(*

## Short summary

This class implements the breadth first iteration strategy for balanced binary search trees.

.. <legal notes>

legal notes
=================
| SPDX-FileCopyrightText: © 2024 ekvip automation GmbH <info@ekvip.de>
| SPDX-License-Identifier: Apache-2.0
| For details check: Apache-2.0_

.. _Apache-2.0: https://www.apache.org/licenses/LICENSE-2.0

.. </legal notes>

*)

{attribute 'enable_dynamic_creation'}
FUNCTION_BLOCK BfsBbstIterator EXTENDS AbstractBalancedBinarySearchTreeIterator

PROPERTY className :CNM_AbstractObject.ClassName
GET
className := 'CNM_Collections.BFS_BBSTIterator';
END_GET
END_PROPERTY

(*

## Short summary

Gets the next Node that iterate should process.

.. <legal notes>

legal notes
=================
| SPDX-FileCopyrightText: © 2022 ekvip automation GmbH <info@ekvip.de>
| SPDX-License-Identifier: Apache-2.0
| For details check: Apache-2.0_

.. _Apache-2.0: https://www.apache.org/licenses/LICENSE-2.0

.. </legal notes>


**Return:** ``TRUE`` a valid node existed, ``FALSE`` no node for iteration existed

*)

METHOD PROTECTED getNextTreeNode : BOOL
VAR_OUTPUT
	node	:CNM_CollectionInterfaces.IBinaryTreeNode;
END_VAR
VAR
	tmpObject :CNM_AbstractObject.IObject;
END_VAR
tmpObject := THIS^.nodeList.dequeue();
__QUERYINTERFACE(tmpObject, node);
getNextTreeNode := THIS^.isObjectValid(node);
END_METHOD

(*

## Short summary

This method appends (if they exists) the left and right child of the node to the nodelist.

.. <legal notes>

legal notes
=================
| SPDX-FileCopyrightText: © 2022 ekvip automation GmbH <info@ekvip.de>
| SPDX-License-Identifier: Apache-2.0
| For details check: Apache-2.0_

.. _Apache-2.0: https://www.apache.org/licenses/LICENSE-2.0

.. </legal notes>



*)

METHOD PROTECTED processNode
VAR_INPUT
	nodeToProcess	: CNM_CollectionInterfaces.IBinaryTreeNode;
END_VAR
IF(nodeToProcess.leftChild <> 0)THEN
	THIS^.nodeList.append(nodeToProcess.leftChild);
END_IF
IF(nodeToProcess.rightChild <> 0)THEN
	THIS^.nodeList.append(nodeToProcess.rightChild);
END_IF
END_METHOD

END_FUNCTION_BLOCK

(* stored: Version 1.1.0.1, ProductVersion 3.1.4026.12
   POU BfsBbstIterator: Id {6aac5e11-1f74-4d52-8b74-0c42fe7b1a2f}, SpecialFunc None
   Property className: Id {d9c15d61-eb3c-459c-ab1c-acd72842ebef}
   Get Get: Id {2235bd85-b217-4725-9bea-f6f4cc955c57}
   Method getNextTreeNode: Id {ebc897b8-539e-41ea-b527-bcfeee98df58}
   Method processNode: Id {26889ffc-74ff-46d2-a1ca-3deb2b839426} *)
